# B&R Automation Studio project Kesim (part 6)

#### Main.st
```iecst
(********************************************************************
 * COPYRIGHT --  B&R Industrial Automation GmbH
 ********************************************************************
 * Task: SUB0
 * Author: kay3a
 * Created: October 16, 2024/11:06 AM
 ********************************************************************
 * Description: Machine CncCtrl task
 ********************************************************************)
PROGRAM _INIT

	//|ŻŻŻŻŻŻŻŻŻŻŻŻŻŻŻŻŻŻŻŻŻŻŻŻŻŻŻŻŻŻŻŻŻŻŻŻŻŻŻŻŻŻŻŻŻŻŻŻŻŻŻŻŻŻŻŻŻŻŻŻŻŻŻŻŻŻŻŻŻŻŻŻŻ
	//|               CNC Klasörünü olustur
	//|_________________________________________________________________________
	Loc.FB.DirCreate.Parameters.DeviceName := 'DEV_CNC';
	Loc.FB.DirCreate.Parameters.DirPath := '/DEVICE=USER_PATH/CNC';
	Loc.FB.DirCreate.Enable := TRUE;
	REPEAT
		Loc.FB.DirCreate.Execute := Loc.FB.DirCreate.Active AND NOT Loc.FB.DirCreate.CommandBusy AND NOT Loc.FB.DirCreate.CommandDone;
		Loc.FB.DirCreate();
		UNTIL Loc.FB.DirCreate.CommandDone
	END_REPEAT;
	//|_________________________________________________________________________

	//|ŻŻŻŻŻŻŻŻŻŻŻŻŻŻŻŻŻŻŻŻŻŻŻŻŻŻŻŻŻŻŻŻŻŻŻŻŻŻŻŻŻŻŻŻŻŻŻŻŻŻŻŻŻŻŻŻŻŻŻŻŻŻŻŻŻŻŻŻŻŻŻŻŻ
	//|               CNC File olustur
	//|_________________________________________________________________________
	Loc.FB.FileCreate.Parameters.DeviceName := 'DEV_CNC';
	Loc.FB.FileCreate.Parameters.FileName := 'Program.cnc';
	Loc.FB.FileCreate.Enable := TRUE;
	REPEAT
		Loc.FB.FileCreate.Execute := Loc.FB.FileCreate.Active AND NOT Loc.FB.FileCreate.CommandBusy AND NOT Loc.FB.FileCreate.CommandDone;
		Loc.FB.FileCreate();
		UNTIL Loc.FB.FileCreate.CommandDone
	END_REPEAT;
	//|_________________________________________________________________________

	//|ŻŻŻŻŻŻŻŻŻŻŻŻŻŻŻŻŻŻŻŻŻŻŻŻŻŻŻŻŻŻŻŻŻŻŻŻŻŻŻŻŻŻŻŻŻŻŻŻŻŻŻŻŻŻŻŻŻŻŻŻŻŻŻŻŻŻŻŻŻŻŻŻŻ
	//|               L I V E    F B s
	//|_________________________________________________________________________
	(* PML *)
	Loc.FB.PML.MpLink := ADR(gMpLink_PackMLSyncModule_CncCtrl);
	Loc.FB.PML.Parameters := ADR(Loc.Par.PML);
	Loc.FB.PML.Enable := TRUE;

	(* CNC *)
	Loc.FB.Cnc3Axis.MpLink := ADR(gMpLink_CncXYZ);
	Loc.FB.Cnc3Axis.Parameters := ADR(Loc.Par.Cnc3Axis);
	Loc.FB.Cnc3Axis.Enable := TRUE;
	Loc.FB.Cnc3Axis.Override := 100.0;
	// Par
	Loc.Par.Cnc3Axis.ProgramName := 'Program.cnc';
	//|_________________________________________________________________________

END_PROGRAM

PROGRAM _CYCLIC

	//|ŻŻŻŻŻŻŻŻŻŻŻŻŻŻŻŻŻŻŻŻŻŻŻŻŻŻŻŻŻŻŻŻŻŻŻŻŻŻŻŻŻŻŻŻŻŻŻŻŻŻŻŻŻŻŻŻŻŻŻŻŻŻŻŻŻŻŻŻŻŻŻŻŻ
	//|                P M L      S T A T E      C U R R E N T
	//|_________________________________________________________________________
	CASE Loc.FB.PML.StateCurrent OF

		//|ŻŻŻŻŻŻŻŻŻŻŻŻŻŻŻŻŻŻŻŻŻŻŻŻŻŻŻŻŻŻŻŻŻŻŻŻŻŻŻŻŻŻŻŻŻŻŻŻŻŻŻŻŻŻŻŻŻŻŻŻŻŻŻŻŻŻŻŻŻŻŻŻŻ
		mpPACKML_STATE_IDLE:	// Idle State
			//|_________________________________________________________________________
			Idle;
			//|_________________________________________________________________________

			//|ŻŻŻŻŻŻŻŻŻŻŻŻŻŻŻŻŻŻŻŻŻŻŻŻŻŻŻŻŻŻŻŻŻŻŻŻŻŻŻŻŻŻŻŻŻŻŻŻŻŻŻŻŻŻŻŻŻŻŻŻŻŻŻŻŻŻŻŻŻŻŻŻŻ
		mpPACKML_STATE_EXECUTE:	// Execute State
			//|_________________________________________________________________________
			Execute;
			//|_________________________________________________________________________

			//|ŻŻŻŻŻŻŻŻŻŻŻŻŻŻŻŻŻŻŻŻŻŻŻŻŻŻŻŻŻŻŻŻŻŻŻŻŻŻŻŻŻŻŻŻŻŻŻŻŻŻŻŻŻŻŻŻŻŻŻŻŻŻŻŻŻŻŻŻŻŻŻŻŻ
		mpPACKML_STATE_COMPLETE:	//
			//|_________________________________________________________________________
			Complete;
			//|_________________________________________________________________________

			//|ŻŻŻŻŻŻŻŻŻŻŻŻŻŻŻŻŻŻŻŻŻŻŻŻŻŻŻŻŻŻŻŻŻŻŻŻŻŻŻŻŻŻŻŻŻŻŻŻŻŻŻŻŻŻŻŻŻŻŻŻŻŻŻŻŻŻŻŻŻŻŻŻŻ
		mpPACKML_STATE_COMPLETING:	// Completing State
			//|_________________________________________________________________________
			Completing;
			//|_________________________________________________________________________

			//|ŻŻŻŻŻŻŻŻŻŻŻŻŻŻŻŻŻŻŻŻŻŻŻŻŻŻŻŻŻŻŻŻŻŻŻŻŻŻŻŻŻŻŻŻŻŻŻŻŻŻŻŻŻŻŻŻŻŻŻŻŻŻŻŻŻŻŻŻŻŻŻŻŻ
		mpPACKML_STATE_STARTING:	// Starting State
			//|_________________________________________________________________________
			Starting;
			//|_________________________________________________________________________

			//|ŻŻŻŻŻŻŻŻŻŻŻŻŻŻŻŻŻŻŻŻŻŻŻŻŻŻŻŻŻŻŻŻŻŻŻŻŻŻŻŻŻŻŻŻŻŻŻŻŻŻŻŻŻŻŻŻŻŻŻŻŻŻŻŻŻŻŻŻŻŻŻŻŻ
		mpPACKML_STATE_SUSPENDED:	//
			//|_________________________________________________________________________
			Suspended;
			//|_________________________________________________________________________

			//|ŻŻŻŻŻŻŻŻŻŻŻŻŻŻŻŻŻŻŻŻŻŻŻŻŻŻŻŻŻŻŻŻŻŻŻŻŻŻŻŻŻŻŻŻŻŻŻŻŻŻŻŻŻŻŻŻŻŻŻŻŻŻŻŻŻŻŻŻŻŻŻŻŻ
		mpPACKML_STATE_HOLDING:	//
			//|_________________________________________________________________________
			Holding;
			//|_________________________________________________________________________

			//|ŻŻŻŻŻŻŻŻŻŻŻŻŻŻŻŻŻŻŻŻŻŻŻŻŻŻŻŻŻŻŻŻŻŻŻŻŻŻŻŻŻŻŻŻŻŻŻŻŻŻŻŻŻŻŻŻŻŻŻŻŻŻŻŻŻŻŻŻŻŻŻŻŻ
		mpPACKML_STATE_HELD:	//
			//|_________________________________________________________________________
			Held;
			//|_________________________________________________________________________

			//|ŻŻŻŻŻŻŻŻŻŻŻŻŻŻŻŻŻŻŻŻŻŻŻŻŻŻŻŻŻŻŻŻŻŻŻŻŻŻŻŻŻŻŻŻŻŻŻŻŻŻŻŻŻŻŻŻŻŻŻŻŻŻŻŻŻŻŻŻŻŻŻŻŻ
		mpPACKML_STATE_UNHOLDING:	//
			//|_________________________________________________________________________
			Unholding;
			//|_________________________________________________________________________

			//|ŻŻŻŻŻŻŻŻŻŻŻŻŻŻŻŻŻŻŻŻŻŻŻŻŻŻŻŻŻŻŻŻŻŻŻŻŻŻŻŻŻŻŻŻŻŻŻŻŻŻŻŻŻŻŻŻŻŻŻŻŻŻŻŻŻŻŻŻŻŻŻŻŻ
		mpPACKML_STATE_SUSPENDING:	//
			//|_________________________________________________________________________
			Suspending;
			//|_________________________________________________________________________

			//|ŻŻŻŻŻŻŻŻŻŻŻŻŻŻŻŻŻŻŻŻŻŻŻŻŻŻŻŻŻŻŻŻŻŻŻŻŻŻŻŻŻŻŻŻŻŻŻŻŻŻŻŻŻŻŻŻŻŻŻŻŻŻŻŻŻŻŻŻŻŻŻŻŻ
		mpPACKML_STATE_UNSUSPENDING:	//
			//|_________________________________________________________________________
			Unsuspending;
			//|_________________________________________________________________________

			//|ŻŻŻŻŻŻŻŻŻŻŻŻŻŻŻŻŻŻŻŻŻŻŻŻŻŻŻŻŻŻŻŻŻŻŻŻŻŻŻŻŻŻŻŻŻŻŻŻŻŻŻŻŻŻŻŻŻŻŻŻŻŻŻŻŻŻŻŻŻŻŻŻŻ
		mpPACKML_STATE_CLEARING:	// Clearing State
			//|_________________________________________________________________________
			Clearing;
			//|_________________________________________________________________________

			//|ŻŻŻŻŻŻŻŻŻŻŻŻŻŻŻŻŻŻŻŻŻŻŻŻŻŻŻŻŻŻŻŻŻŻŻŻŻŻŻŻŻŻŻŻŻŻŻŻŻŻŻŻŻŻŻŻŻŻŻŻŻŻŻŻŻŻŻŻŻŻŻŻŻ
		mpPACKML_STATE_STOPPED:	//
			//|_________________________________________________________________________
			Stopped;
			//|_________________________________________________________________________

			//|ŻŻŻŻŻŻŻŻŻŻŻŻŻŻŻŻŻŻŻŻŻŻŻŻŻŻŻŻŻŻŻŻŻŻŻŻŻŻŻŻŻŻŻŻŻŻŻŻŻŻŻŻŻŻŻŻŻŻŻŻŻŻŻŻŻŻŻŻŻŻŻŻŻ
		mpPACKML_STATE_STOPPING:	// Stopping State
			//|_________________________________________________________________________
			Stopping;
			//|_________________________________________________________________________

			//|ŻŻŻŻŻŻŻŻŻŻŻŻŻŻŻŻŻŻŻŻŻŻŻŻŻŻŻŻŻŻŻŻŻŻŻŻŻŻŻŻŻŻŻŻŻŻŻŻŻŻŻŻŻŻŻŻŻŻŻŻŻŻŻŻŻŻŻŻŻŻŻŻŻ
		mpPACKML_STATE_ABORTING:	// Aborting State
			//|_________________________________________________________________________
			Aborting;
			//|_________________________________________________________________________

			//|ŻŻŻŻŻŻŻŻŻŻŻŻŻŻŻŻŻŻŻŻŻŻŻŻŻŻŻŻŻŻŻŻŻŻŻŻŻŻŻŻŻŻŻŻŻŻŻŻŻŻŻŻŻŻŻŻŻŻŻŻŻŻŻŻŻŻŻŻŻŻŻŻŻ
		mpPACKML_STATE_ABORTED:	//
			//|_________________________________________________________________________
			Aborted;
			//|_________________________________________________________________________

			//|ŻŻŻŻŻŻŻŻŻŻŻŻŻŻŻŻŻŻŻŻŻŻŻŻŻŻŻŻŻŻŻŻŻŻŻŻŻŻŻŻŻŻŻŻŻŻŻŻŻŻŻŻŻŻŻŻŻŻŻŻŻŻŻŻŻŻŻŻŻŻŻŻŻ
		mpPACKML_STATE_RESETTING:	// Resetting State
			//|_________________________________________________________________________
			Resetting;
			//|_________________________________________________________________________

			//|ŻŻŻŻŻŻŻŻŻŻŻŻŻŻŻŻŻŻŻŻŻŻŻŻŻŻŻŻŻŻŻŻŻŻŻŻŻŻŻŻŻŻŻŻŻŻŻŻŻŻŻŻŻŻŻŻŻŻŻŻŻŻŻŻŻŻŻŻŻŻŻŻŻ
		ELSE	// All state which are not defined are handled in this part.
			//|_________________________________________________________________________
			Loc.FB.PML.Command.StateComplete := TRUE;
			//|_________________________________________________________________________

	END_CASE;
	//|_________________________________________________________________________

	//|ŻŻŻŻŻŻŻŻŻŻŻŻŻŻŻŻŻŻŻŻŻŻŻŻŻŻŻŻŻŻŻŻŻŻŻŻŻŻŻŻŻŻŻŻŻŻŻŻŻŻŻŻŻŻŻŻŻŻŻŻŻŻŻŻŻŻŻŻŻŻŻŻŻ
	//|              C A L L    F B s
	//|_________________________________________________________________________
	(* PML *)
	Loc.FB.PML();

	(* Axis *)
	Loc.FB.Cnc3Axis();
	//|_________________________________________________________________________

END_PROGRAM

PROGRAM _EXIT

	//|ŻŻŻŻŻŻŻŻŻŻŻŻŻŻŻŻŻŻŻŻŻŻŻŻŻŻŻŻŻŻŻŻŻŻŻŻŻŻŻŻŻŻŻŻŻŻŻŻŻŻŻŻŻŻŻŻŻŻŻŻŻŻŻŻŻŻŻŻŻŻŻŻŻ
	//|              K I L L   F B s
	//|_________________________________________________________________________
	(* PML *)
	Loc.FB.PML(Enable := FALSE);

	(* CNC *)
	Loc.FB.Cnc3Axis(Enable := FALSE);
	//|_________________________________________________________________________

END_PROGRAM
```

#### Program Logical/Source/CncCtrl/act_PML/Unused

##### Holding.st
```iecst
(*********************************************************************************
 * Copyright: B&R Industrial Automation GmbH
 * Author:    kay3a
 * Created:   June 21, 2023/5:55 PM
 *********************************************************************************)
ACTION Holding:

	Loc.FB.PML.Command.StateComplete := TRUE;

END_ACTION
```

#### Program Logical/Source/CncCtrl/act_PML/Used

##### Aborted.st
```iecst
(*********************************************************************************
 * Copyright: B&R Industrial Automation GmbH
 * Author:    kay3a
 * Created:   June 21, 2023/5:55 PM
 *********************************************************************************)
ACTION Aborted:

END_ACTION
```

##### Aborting.st
```iecst
(*********************************************************************************
 * Copyright: B&R Industrial Automation GmbH
 * Author:    kay3a
 * Created:   June 21, 2023/5:55 PM
 *********************************************************************************)
ACTION Aborting:

Loc.FB.PML.Command.StateComplete := TRUE;

END_ACTION
```

##### Clearing.st
```iecst
(*********************************************************************************
 * Copyright: B&R Industrial Automation GmbH
 * Author:    kay3a
 * Created:   June 21, 2023/5:55 PM
 *********************************************************************************)
ACTION Clearing:

	Loc.FB.PML.Command.StateComplete := TRUE;

END_ACTION
```

##### Resetting.st
```iecst
(*********************************************************************************
 * Copyright: B&R Industrial Automation GmbH
 * Author:    kay3a
 * Created:   June 21, 2023/5:55 PM
 *********************************************************************************)
ACTION Resetting:

Loc.FB.PML.Command.StateComplete := TRUE;

END_ACTION
```

##### Stopped.st
```iecst
(*********************************************************************************
 * Copyright: B&R Industrial Automation GmbH
 * Author:    kay3a
 * Created:   June 21, 2023/5:55 PM
 *********************************************************************************)
ACTION Stopped:

END_ACTION
```

##### Suspending.st
```iecst
(*********************************************************************************
 * Copyright: B&R Industrial Automation GmbH
 * Author:    kay3a
 * Created:   June 21, 2023/5:55 PM
 *********************************************************************************)
ACTION Suspending:

Loc.FB.PML.Command.StateComplete := TRUE;

END_ACTION
```

##### Unsuspending.st
```iecst
(*********************************************************************************
 * Copyright: B&R Industrial Automation GmbH
 * Author:    kay3a
 * Created:   June 21, 2023/5:55 PM
 *********************************************************************************)
ACTION Unsuspending:

	Loc.FB.PML.Command.StateComplete := TRUE;

END_ACTION
```

### Variables.var
```iecst
(********************************************************************
 * COPYRIGHT --  B&R Industrial Automation GmbH
 *******************************************************************
 * Task: AlarmX
 * Author: kay3a
 * Created: October 2, 2024/3:55 PM
 ********************************************************************)
(**)
(**** Local variables*)
VAR
	Loc : Loc_typ; (**** Bu Task icinde kullanilacak Local degisken*)
END_VAR
(**)
```

### Constants.var
```iecst
(********************************************************************
 * COPYRIGHT --  B&R Industrial Automation GmbH
 *******************************************************************
 * Task: UserX
 * Author: kay3a
 * Created: October 2, 2024/3:55 PM
 ********************************************************************)
(**)
(**** Alarm Category Constants*)
VAR CONSTANT
	USER_LIST_MAX_SELECTION : USINT := 20; (*Maxiumum selections on the User List *)
	USER_LIST_RANGE_START : USINT := 0; (*Range start (used for UserXMgrUIConnect)*)
	USER_LIST_RANGE_END : USINT := 20; (*Range end (used for UserXMgrUIConnect)*)
END_VAR
```

Listed in the project but not available here: Logical/Libraries/CMS_CT/Constants.var, Logical/SourceCode/MAIN/Exit.st, Logical/SourceCode/CncCtrl/act_PML/Used/Resetting.st, Logical/SourceCode/CncCtrl/act_PML/Used/Clearing.st, Logical/SourceCode/CncCtrl/act_PML/Used/Aborting.st, Logical/SourceCode/CncCtrl/act_PML/Used/Suspending.st, Logical/SourceCode/CncCtrl/act_PML/Used/Unsuspending.st, Logical/SourceCode/CncCtrl/act_PML/Used/Aborted.st, Logical/SourceCode/CncCtrl/act_PML/Used/Stopped.st, Logical/SourceCode/CncCtrl/act_PML/Unused/Holding.st, Logical/SourceCode/Infastructure/AlarmX/Variables.var, Logical/SourceCode/Infastructure/AlarmX/Constants.var, Logical/SourceCode/Infastructure/UserXMgr/Types.typ, Logical/SourceCode/Infastructure/UserXMgr/Constants.var, Logical/SourceCode/Infastructure/UserXMgr/HMIAction.st, Logical/CuttingTable/RecipeHandling/Types.typ
